Omron CX-Programmer project NewProject (CX-Programmer 9.61)

# PLC traficlight: CP1E N30

## Global symbols (name address type ; comment)
0.00 BOOL  ; STOP
0.01 BOOL  ; START
100.00 BOOL  ; LAMPU MERAH
100.01 BOOL  ; LAMPU KUNING
100.02 BOOL  ; LAMPU HIJAU
5.00 BOOL  ; IR
T001 BOOL  ; WAKTU 1
T002 BOOL  ; WAKTU 2
T003 BOOL  ; WAKTU 3

## Program NewProgram1 (cyclic task 0)
Local symbols
END BOOL

### Section Section1

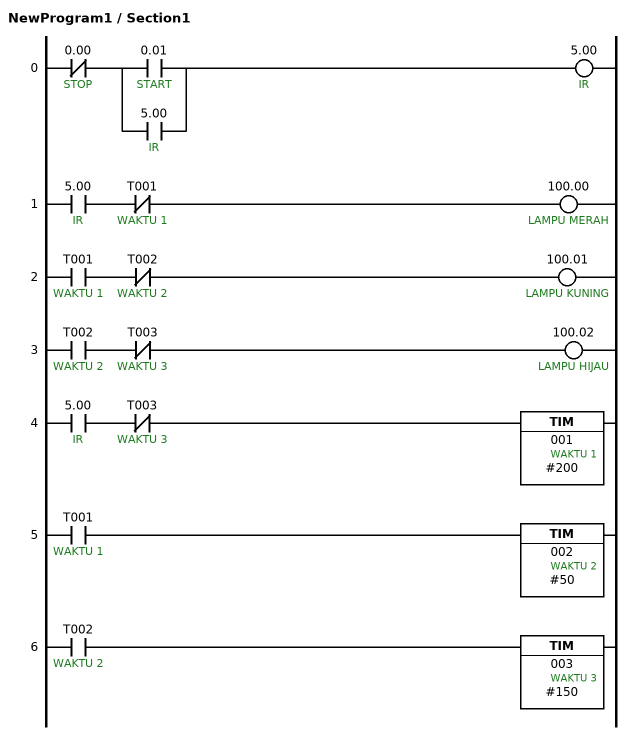
; rung 0
LDNOT 0.00  ; STOP
LD 0.01  ; START
OR 5.00  ; IR
ANDLD
OUT 5.00  ; IR
; rung 1
LD 5.00  ; IR
ANDNOT T001  ; WAKTU 1
OUT 100.00  ; LAMPU MERAH
; rung 2
LD T001  ; WAKTU 1
ANDNOT T002  ; WAKTU 2
OUT 100.01  ; LAMPU KUNING
; rung 3
LD T002  ; WAKTU 2
ANDNOT T003  ; WAKTU 3
OUT 100.02  ; LAMPU HIJAU
; rung 4
LD 5.00  ; IR
ANDNOT T003  ; WAKTU 3
TIM 001 #200  ; WAKTU 1
; rung 5
LD T001  ; WAKTU 1
TIM 002 #50  ; WAKTU 2
; rung 6
LD T002  ; WAKTU 2
TIM 003 #150  ; WAKTU 3
; rung 7
END(001)

### Section END
; rung 0
END(001)